Universal Robots URScript: Program_Control_MoveJ.script

def Program_Template():
   set_standard_analog_input_domain(0, 1)
   set_standard_analog_input_domain(1, 1)
   set_tool_analog_input_domain(0, 1)
   set_tool_analog_input_domain(1, 1)
   set_analog_outputdomain(0, 0)
   set_analog_outputdomain(1, 0)
   set_tool_voltage(0)
   set_input_actions_to_default()
   set_tcp(p[0.0,0.0,0.0,0.0,0.0,0.0])
   set_payload(0.0)
   set_gravity([0.0, 0.0, 9.82])
   global Base=p[0.0,0.0,0.0,0.0,0.0,0.0]
   rtde_set_watchdog("speed_slider_mask", 10.0, "ignore")
   global setp = [0,0,0,0,0,0]
   global move = [0,0,0,0]


   thread Update():
      setp = get_actual_joint_positions()

      while True:

         tmp = [0,0,0,0,0,0]
         tmp[0] = read_input_float_register(0)
         tmp[1] = read_input_float_register(1)
         tmp[2] = read_input_float_register(2)
         tmp[3] = read_input_float_register(3)
         tmp[4] = read_input_float_register(4)
         tmp[5] = read_input_float_register(5)

         move = [0,0,0,0]
         move[0] = read_input_float_register(6)
         move[1] = read_input_float_register(7)
         move[2] = read_input_float_register(8)
         move[3] = read_input_float_register(9)

         setp = tmp

         sync()

      end
   end

   textmsg("Listening for MoveJ")

   write_output_integer_register(0, 0)
   run Update()

   if read_input_integer_register(1)!=1:

      textmsg("Input Int Register 1 is not reset! Value = ",read_input_integer_register(1))
      textmsg("Input Int Register 0 value = ",read_input_integer_register(0))

      i = 0
      while i < 10:
         textmsg(i,read_input_float_register(i))
         i = i+1
      end
   end

   setp = get_actual_joint_positions()
   rtde_set_watchdog("input_int_register_0",1,"PAUSE")

   while read_input_integer_register(1)==1:
      write_output_integer_register(0, 0)
      sync()

      movej( setp, move[0] , move[1], move[2], move[3])

      write_output_integer_register(0, 1)
      sync()
  end

  textmsg("Ending MoveJ")

  write_output_integer_register(0, 0)


end
